// Implicitly generated code : DO NOT EDIT
FUNCTION CheckLRangeUnsigned : ULINT
VAR_INPUT
	value, lower, upper: ULINT;
END_VAR

// Implicitly generated code : Only an Implementation suggestion
{noflow}
IF (value < lower) THEN
	CheckLRangeUnsigned := lower;
ELSIF(value > upper) THEN
	CheckLRangeUnsigned := upper;
ELSE
	CheckLRangeUnsigned := value;
END_IF
{flow}

END_FUNCTION

(* stored: Version 1.1.0.1, ProductVersion 3.1.4024.2
   POU CheckLRangeUnsigned: Id {0eeff54e-a32a-4bdc-a09d-5dd3ad7769c1}, SpecialFunc CheckLRangeUnsigned *)
